INTERFACE I_Event EXTENDS __SYSTEM.IQueryInterface

END_INTERFACE

(* stored: Version 1.1.0.1, ProductVersion 3.1.4024.12
   Itf I_Event: Id {6c00c587-90f8-0715-3019-8fe4305f1f00} *)
